(* CoDeSys 2.3 export: CALCVOLTAGETOMOTORVAL.EXP *)

(* POU \/calcVoltageToMotorVal, ST *)
FUNCTION calcVoltageToMotorVal : INT
VAR_INPUT
    r_voltage : REAL;
END_VAR
VAR
    r_MotorVoltage : REAL := FALSE;
END_VAR
calcVoltageToMotorVal := (32767.0 / r_MotorVoltage.0) * r_voltage;
END_FUNCTION
